// TIA Portal V19 export
TYPE "C701_VAR_IF_VAT_BUF_TYPIC"
   STRUCT
      STO { ExternalAccessible := 'False'; ExternalVisible := 'False'; ExternalWritable := 'False'} : Struct   // Opsomming van alle storingen
         A001 : Bool;   // Fout temperatuurmeting in vertrek
         A002 : Bool;   // Fout temperatuurmeting uit vertrek
         A003 : Bool;   // Fout temperatuurmeting in retour
         A004 : Bool;   // Fout temperatuurmeting uit retour
      END_STRUCT;
   END_STRUCT;
END_TYPE
